TYPE DUT_SENSOR_DATAS_h6 :
UNION
	data_lreal:REAL;
	data_byte:ARRAY[0..3] OF BYTE;
END_UNION
END_TYPE

(* stored: Version 1.1.0.1, ProductVersion 3.1.4024.6
   DUT DUT_SENSOR_DATAS_h6: Id {b82c6200-4d6d-4347-91ed-859ceb05f790} *)
